Staubli VAL3: prdMassage.pgx

program prdMassage()
  local num l_nNum
begin
  do

    //call $rotAngle()
    //生产中,数据读取中
    if read:bCycle and !read:bWriteEnd
      //路径加载中
      if roundDown(read:nMoveID)>read:nWritePtr+read:nThousandWrite*1000
        call massage("等待路径加载...")
      else
        if bPause
          if bInterVal
            call massage("间断恢复:"+toString(".1",nPauseTime-(clock()-nTimeBuff))+"秒")
          else
            call massage("暂停中,按F3继续生产")
          endIf
        else
          call massage("生产中,等待生产结束")
        endIf
      endIf
      //生产中,数据读取结束
    elseIf read:bCycle and read:bWriteEnd
      if bPause
        if bInterVal
          call massage("间断恢复:"+toString(".1",nPauseTime-(clock()-nTimeBuff))+"秒")
        else
          call massage("暂停中,按F3继续生产")
        endIf
      else
        call massage("生产中,等待生产结束")
      endIf
      //生产结束
    elseIf read:bCycle==false and read:bCycleEnd==true
      call massage("生产结束")
    endIf
    delay(0)
  until read:bCycle==false and read:bCycleEnd==true
  call massage("生产结束")
end
